(* IEC 61131-3 sources: verifaps-lib/geteta/examples/constantprogram, 1 file *)

(* ---- constantprogram.st ---- *)
PROGRAM constantprogram
    VAR_INPUT
        i : INT;
    END_VAR

    VAR_OUTPUT
        o : INT;
        c : INT;
    END_VAR

    o := i;
    c := 42;

END_PROGRAM
